Omron CX-Programmer project NewProject (CX-Programmer 9.63)

# PLC AutoAvanPLC: CJ2M CPU33
I/O table (CPU CJ2M-CPU33): rack 0 slot 0 CJ1W-ID211; rack 0 slot 1 CJ1W-OC211; rack 0 slot 11 CJ2M-EIP21

## Global symbols (name address type ; comment)
AM_ProcStatus W11 CHANNEL  ; Automatic Mode Process Status
AM_SReset W101.01 BOOL  ; Automatic Mode Shift Reset
AM_Shift W100.00 BOOL  ; Automatic Mode Shift
D22.03 BOOL  ; External Out Cilinder
W11.04 BOOL  ; .
B_Start 0.01 BOOL  ; Fisical  Start Button
C_Actual_X D14 CHANNEL  ; Actual X Postion
C_Actual_Y D15 CHANNEL  ; Actual Y Poistion
C_Clock W1.07 BOOL  ; Clock For Cartesian
C_Enable 1.06 BOOL
C_Error 0.07 BOOL  ; Fisical Cartesian Error
C_Next_X D10 CHANNEL  ; New X Position
C_Next_Y D11 CHANNEL  ; Next Y
C_Reach 0.08 BOOL  ; Fisical Cartesian Position Reached
Cartesian CartesianSimulator
DN_Pointer D97 CHANNEL  ; Pointer to the Number of Drills of Program
Drill 1.05 BOOL  ; Fisical Drill
EMERG 0.00 BOOL  ; Fisical Emergency
Ext_CEnable D22.06 BOOL  ; External Cartesian Enable
Ext_Drill D22.05 BOOL  ; External Dril
Ext_GL D22.02 BOOL  ; External Green Light
Ext_RL D22.00 BOOL  ; External Red Light
Ext_YL D22.01 BOOL  ; External Yellow Light
Ext_ZC D22.04 BOOL  ; External Z Cinder
F_AM D20.06 BOOL  ; Flag Automatic Mode
F_EM D20.07 BOOL  ; Flag End Mode
F_Incialization D20.00 BOOL  ; Flag for Incialization Process
F_MM D20.04 BOOL  ; Flag Manual Mode
F_MS D20.02 BOOL  ; Flag for Mode Selection
GL 1.02 BOOL  ; Fisical Green Light
INI_SReset W100.01 BOOL  ; Inicialization Shift Reset
INI_Shift W100.00 BOOL  ; INicialization Shift Bit
I_BStart D0.01 BOOL  ; Start Button
I_CError D0.07 BOOL  ; Cartesian Error
I_CReach D0.08 BOOL  ; Cartesian Position Reached
I_EMERG D0.00 BOOL  ; Emergency
I_SP D0.02 BOOL  ; Piece Sensor
I_a0 D0.03 BOOL  ; Z- Sensor
I_a1 D0.04 BOOL  ; Z+ Sensor
I_a2 D0.05 BOOL  ; O- Sensor
I_a3 D0.06 BOOL  ; O+ Sensor
Init_ProcStatus W10 CHANNEL  ; Inicialization Process status
Init_St0 W10.00 BOOL  ; Inicialization Stage 0
Init_St1 W10.01 BOOL  ; Inicialization Stage 1
Init_St2 W10.02 BOOL  ; Inicialization Stage 2
Init_St3 W10.03 BOOL  ; Inicialization Stage 3
M_Aux W20.01 BOOL  ; Main Process Auxiliary Flag
N_Drills D96 CHANNEL  ; Number of Drill Done
OC 1.03 BOOL  ; Fisical Out Cilinder +
O_CEnable D1.06 BOOL  ; Enable Cartesian Motor
O_Drill D1.05 BOOL  ; Drill
O_GL D1.02 BOOL  ; Green Light
O_OC D1.03 BOOL  ; Out Cilinder +
O_RL D1.00 BOOL  ; Red Light
O_YL D1.01 BOOL  ; Yellow Light
O_ZC D1.04 BOOL  ; Z Cilinder +
PN_Pointer D50 CHANNEL  ; Program Number_Pointer
RL 1.00 BOOL  ; Fisical Red Light
S_P 0.02 BOOL  ; Fisical Piece Sensor
Sct_Auto D20.05 BOOL  ; Selector Automatic Mode
Sct_Manual D20.03 BOOL  ; Select Manual Mode
Sim_C_Reach W1.00 BOOL  ; Simulation of C_Reach
StopNow W0.00 BOOL  ; StopNow
X_Pointer D98 CHANNEL  ; Pointer of Position X
YL 1.01 BOOL  ; Fisical Yellow Light
Y_Pointer D99 CHANNEL  ; Pointer of Position Y
ZC 1.04 BOOL  ; Fisical Z Cilinder +
a_0 0.03 BOOL  ; Fisical Z- Sensor
a_1 0.04 BOOL  ; Fisical Z+ Sensor
a_2 0.05 BOOL  ; Fisical O- Sensor
a_3 0.06 BOOL  ; Fisical O+ Sensor

## Program Auto_Fura (cyclic task 0)
; Auto Fura
Local symbols
DH100 CHANNEL

### Section HWInput_Output

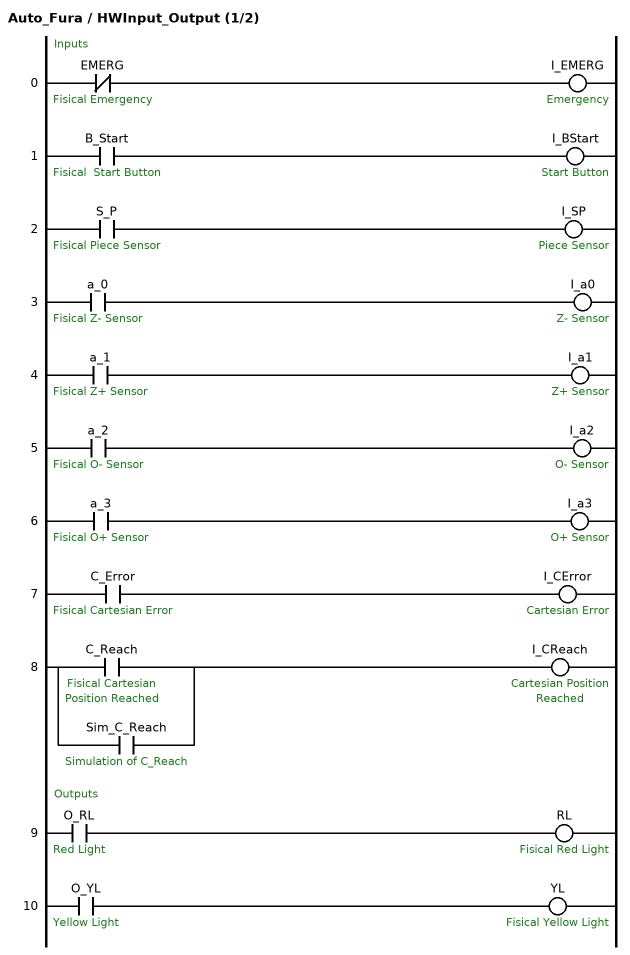
; rung 0: Inputs
LDNOT EMERG  ; Fisical Emergency
OUT I_EMERG  ; Emergency
; rung 1
LD B_Start  ; Fisical  Start Button
OUT I_BStart  ; Start Button
; rung 2
LD S_P  ; Fisical Piece Sensor
OUT I_SP  ; Piece Sensor
; rung 3
LD a_0  ; Fisical Z- Sensor
OUT I_a0  ; Z- Sensor
; rung 4
LD a_1  ; Fisical Z+ Sensor
OUT I_a1  ; Z+ Sensor
; rung 5
LD a_2  ; Fisical O- Sensor
OUT I_a2  ; O- Sensor
; rung 6
LD a_3  ; Fisical O+ Sensor
OUT I_a3  ; O+ Sensor
; rung 7
LD C_Error  ; Fisical Cartesian Error
OUT I_CError  ; Cartesian Error
; rung 8
LD C_Reach  ; Fisical Cartesian Position Reached
OR Sim_C_Reach  ; Simulation of C_Reach
OUT I_CReach  ; Cartesian Position Reached
; rung 9: Outputs
LD O_RL  ; Red Light
OUT RL  ; Fisical Red Light
; rung 10
LD O_YL  ; Yellow Light
OUT YL  ; Fisical Yellow Light

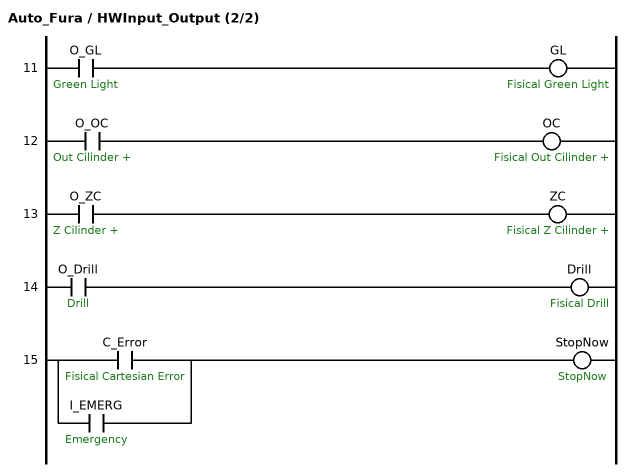
; rung 11
LD O_GL  ; Green Light
OUT GL  ; Fisical Green Light
; rung 12
LD O_OC  ; Out Cilinder +
OUT OC  ; Fisical Out Cilinder +
; rung 13
LD O_ZC  ; Z Cilinder +
OUT ZC  ; Fisical Z Cilinder +
; rung 14
LD O_Drill  ; Drill
OUT Drill  ; Fisical Drill
; rung 15
LD C_Error  ; Fisical Cartesian Error
OR I_EMERG  ; Emergency
OUT StopNow  ; StopNow

### Section Main

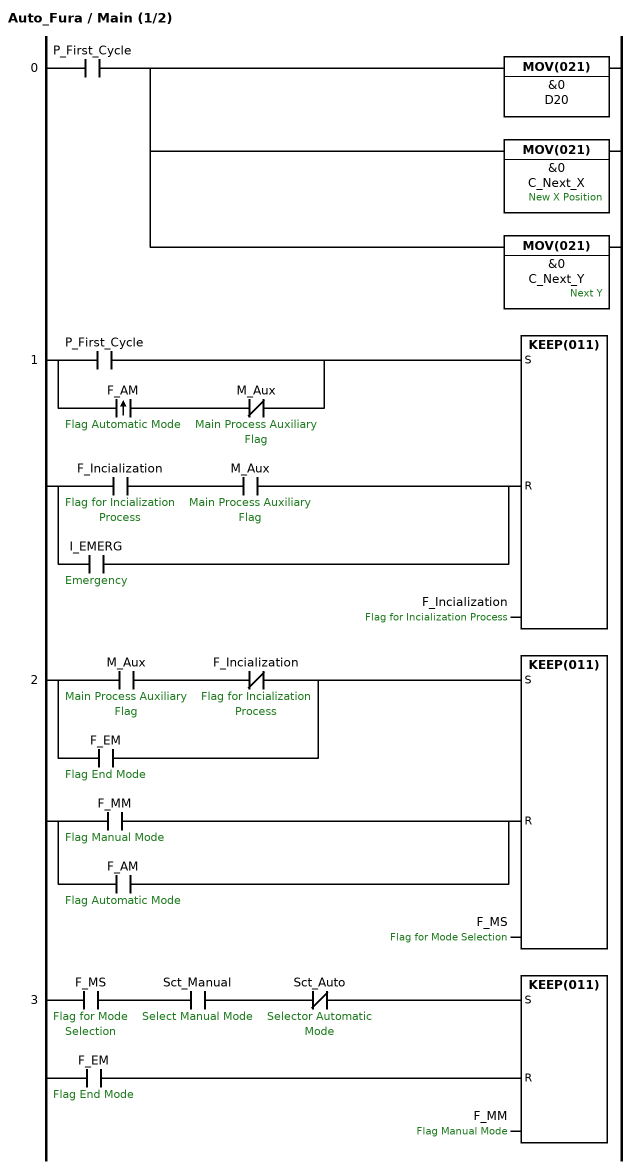
; rung 0
LD P_First_Cycle
MOV(021) &0 D20
MOV(021) &0 C_Next_X  ; New X Position
MOV(021) &0 C_Next_Y  ; Next Y
; rung 1
LD P_First_Cycle
@LD F_AM  ; Flag Automatic Mode
ANDNOT M_Aux  ; Main Process Auxiliary Flag
ORLD
LD F_Incialization  ; Flag for Incialization Process
AND M_Aux  ; Main Process Auxiliary Flag
OR I_EMERG  ; Emergency
KEEP(011) F_Incialization  ; Flag for Incialization Process
; rung 2
LD M_Aux  ; Main Process Auxiliary Flag
ANDNOT F_Incialization  ; Flag for Incialization Process
OR F_EM  ; Flag End Mode
LD F_MM  ; Flag Manual Mode
OR F_AM  ; Flag Automatic Mode
KEEP(011) F_MS  ; Flag for Mode Selection
; rung 3
LD F_MS  ; Flag for Mode Selection
AND Sct_Manual  ; Select Manual Mode
ANDNOT Sct_Auto  ; Selector Automatic Mode
LD F_EM  ; Flag End Mode
KEEP(011) F_MM  ; Flag Manual Mode

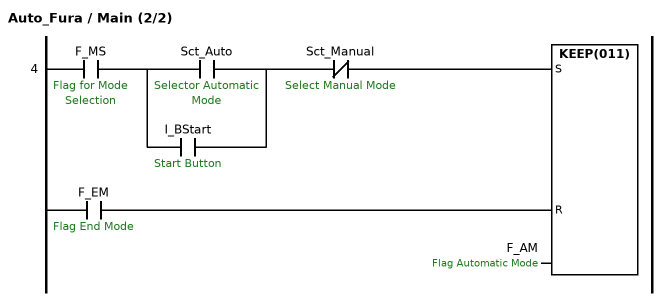
; rung 4
LD F_MS  ; Flag for Mode Selection
LD Sct_Auto  ; Selector Automatic Mode
OR I_BStart  ; Start Button
ANDLD
ANDNOT Sct_Manual  ; Select Manual Mode
LD F_EM  ; Flag End Mode
KEEP(011) F_AM  ; Flag Automatic Mode

### Section Iniciation

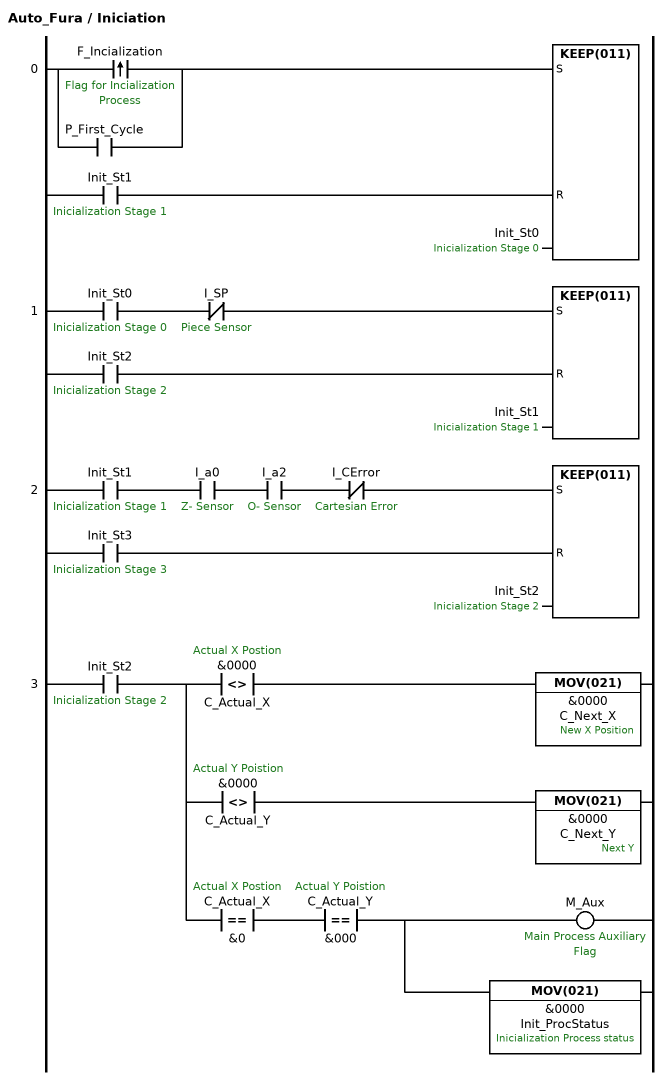
; rung 0
@LD F_Incialization  ; Flag for Incialization Process
OR P_First_Cycle
LD Init_St1  ; Inicialization Stage 1
KEEP(011) Init_St0  ; Inicialization Stage 0
; rung 1
LD Init_St0  ; Inicialization Stage 0
ANDNOT I_SP  ; Piece Sensor
LD Init_St2  ; Inicialization Stage 2
KEEP(011) Init_St1  ; Inicialization Stage 1
; rung 2
LD Init_St1  ; Inicialization Stage 1
AND I_a0  ; Z- Sensor
AND I_a2  ; O- Sensor
ANDNOT I_CError  ; Cartesian Error
LD Init_St3  ; Inicialization Stage 3
KEEP(011) Init_St2  ; Inicialization Stage 2
; rung 3
LD Init_St2  ; Inicialization Stage 2
OUT TR0
AND<>(305) &0000 C_Actual_X  ; Actual X Postion
MOV(021) &0000 C_Next_X  ; New X Position
LD TR0
AND<>(305) &0000 C_Actual_Y  ; Actual Y Poistion
MOV(021) &0000 C_Next_Y  ; Next Y
LD TR0
AND=(300) C_Actual_X &0  ; Actual X Postion
AND=(300) C_Actual_Y &000  ; Actual Y Poistion
OUT M_Aux  ; Main Process Auxiliary Flag
MOV(021) &0000 Init_ProcStatus  ; Inicialization Process status

### Section SerialCam
; Input from Camera

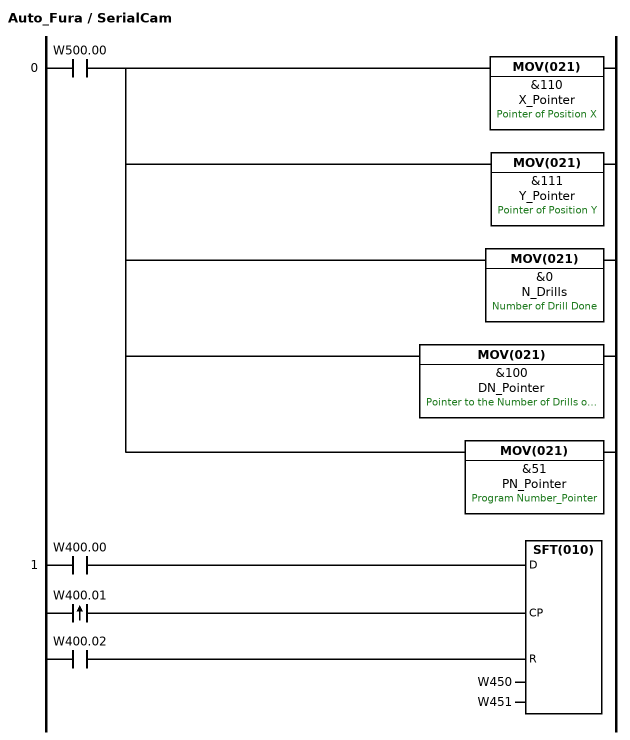
; rung 0
LD W500.00
MOV(021) &110 X_Pointer  ; Pointer of Position X
MOV(021) &111 Y_Pointer  ; Pointer of Position Y
MOV(021) &0 N_Drills  ; Number of Drill Done
MOV(021) &100 DN_Pointer  ; Pointer to the Number of Drills of Program
MOV(021) &51 PN_Pointer  ; Program Number_Pointer
; rung 1
LD W400.00
@LD W400.01
LD W400.02
SFT(010) W450 W451

### Section AutoMode

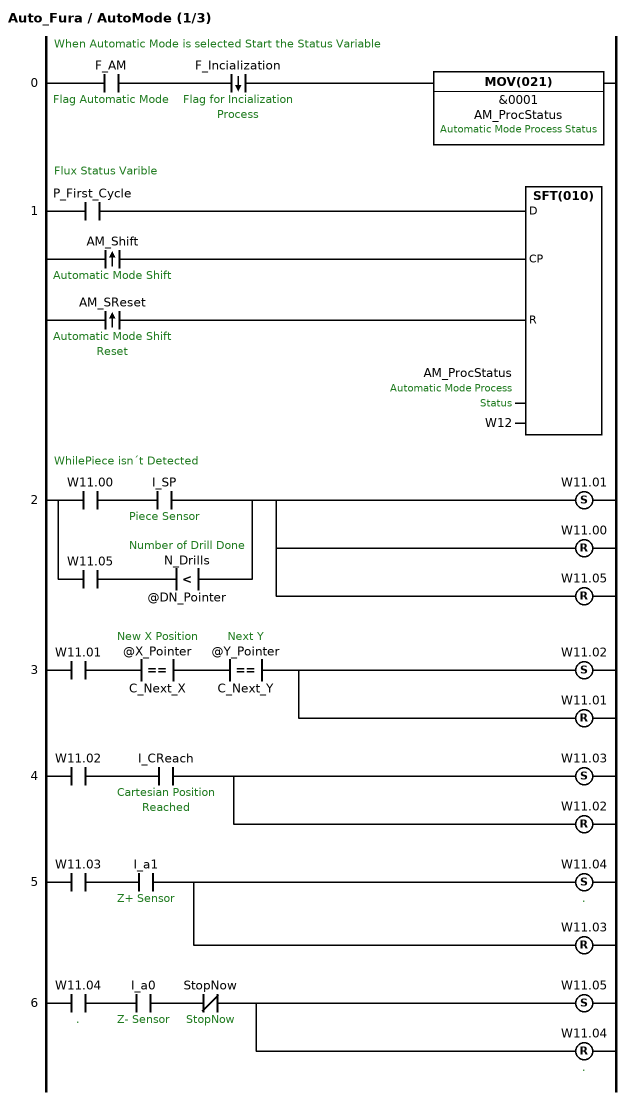
; rung 0: When Automatic Mode is selected Start the Status Variable
LD F_AM  ; Flag Automatic Mode
%AND F_Incialization  ; Flag for Incialization Process
MOV(021) &0001 AM_ProcStatus  ; Automatic Mode Process Status
; rung 1: Flux Status Varible
LD P_First_Cycle
@LD AM_Shift  ; Automatic Mode Shift
@LD AM_SReset  ; Automatic Mode Shift Reset
SFT(010) AM_ProcStatus W12  ; Automatic Mode Process Status
; rung 2: WhilePiece isn´t Detected
LD W11.00
AND I_SP  ; Piece Sensor
LD W11.05
AND<(310) N_Drills @DN_Pointer  ; Number of Drill Done
ORLD
SET W11.01
RSET W11.00
RSET W11.05
; rung 3
LD W11.01
AND=(300) @X_Pointer C_Next_X  ; New X Position
AND=(300) @Y_Pointer C_Next_Y  ; Next Y
SET W11.02
RSET W11.01
; rung 4
LD W11.02
AND I_CReach  ; Cartesian Position Reached
SET W11.03
RSET W11.02
; rung 5
LD W11.03
AND I_a1  ; Z+ Sensor
SET W11.04  ; .
RSET W11.03
; rung 6
LD W11.04  ; .
AND I_a0  ; Z- Sensor
ANDNOT StopNow  ; StopNow
SET W11.05
RSET W11.04  ; .

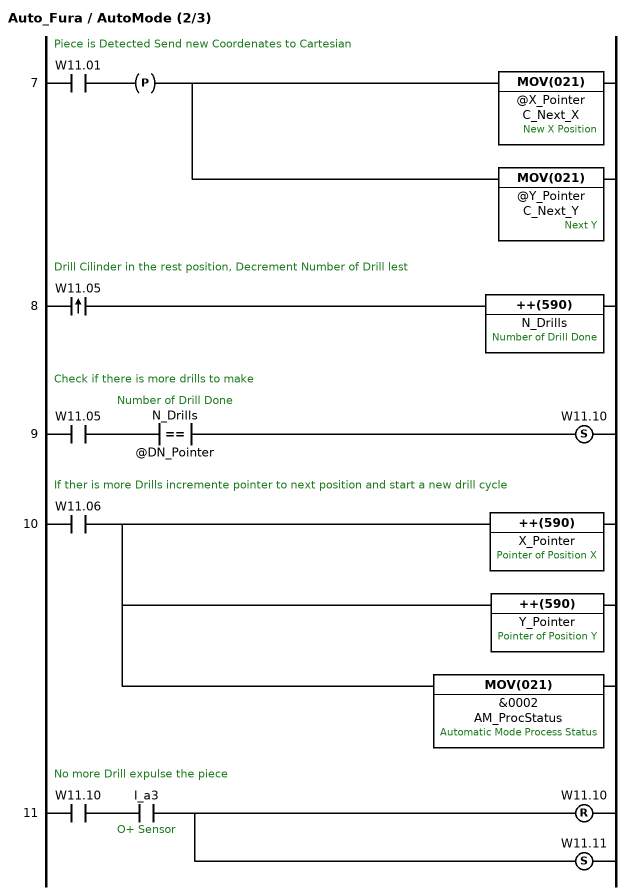
; rung 7: Piece is Detected Send new Coordenates to Cartesian
LD W11.01
UP(521)
MOV(021) @X_Pointer C_Next_X  ; New X Position
MOV(021) @Y_Pointer C_Next_Y  ; Next Y
; rung 8: Drill Cilinder in the rest position, Decrement Number of Drill lest
@LD W11.05
++(590) N_Drills  ; Number of Drill Done
; rung 9: Check if there is more drills to make
LD W11.05
AND=(300) N_Drills @DN_Pointer  ; Number of Drill Done
SET W11.10
; rung 10: If ther is more Drills incremente pointer to next position and start a new drill cycle
LD W11.06
++(590) X_Pointer  ; Pointer of Position X
++(590) Y_Pointer  ; Pointer of Position Y
MOV(021) &0002 AM_ProcStatus  ; Automatic Mode Process Status
; rung 11: No more Drill expulse the piece
LD W11.10
AND I_a3  ; O+ Sensor
RSET W11.10
SET W11.11

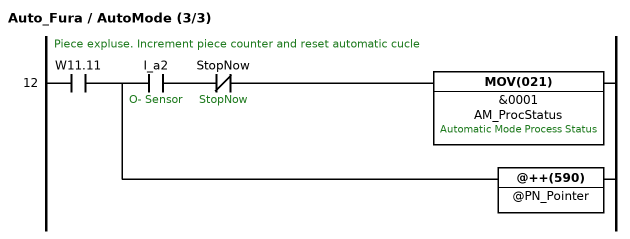
; rung 12: Piece expluse. Increment piece counter and reset automatic cucle
LD W11.11
OUT TR0
AND I_a2  ; O- Sensor
ANDNOT StopNow  ; StopNow
MOV(021) &0001 AM_ProcStatus  ; Automatic Mode Process Status
LD TR0
@++(590) @PN_Pointer

### Section ManualMode

### Section Output

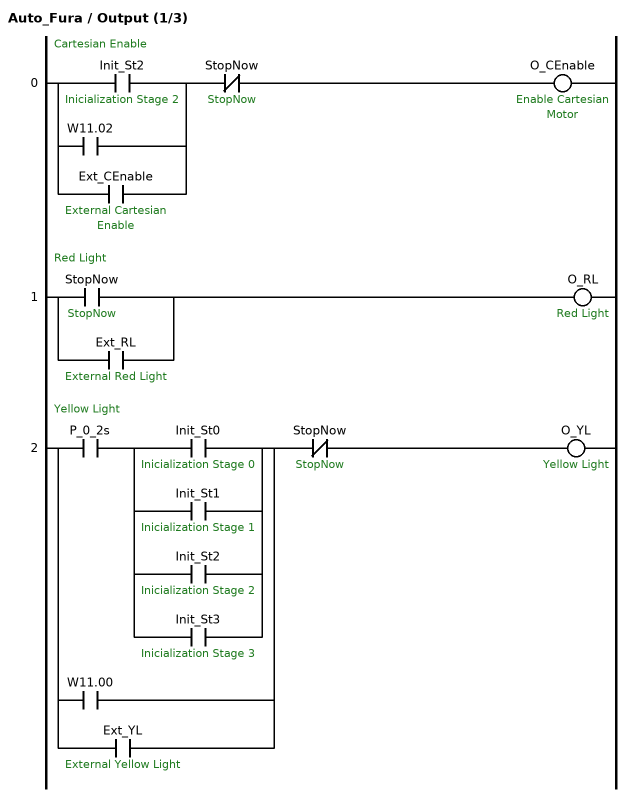
; rung 0: Cartesian Enable
LD Init_St2  ; Inicialization Stage 2
OR W11.02
OR Ext_CEnable  ; External Cartesian Enable
ANDNOT StopNow  ; StopNow
OUT O_CEnable  ; Enable Cartesian Motor
; rung 1: Red Light
LD StopNow  ; StopNow
OR Ext_RL  ; External Red Light
OUT O_RL  ; Red Light
; rung 2: Yellow Light
LD P_0_2s
LD Init_St0  ; Inicialization Stage 0
OR Init_St1  ; Inicialization Stage 1
OR Init_St2  ; Inicialization Stage 2
OR Init_St3  ; Inicialization Stage 3
ANDLD
OR W11.00
OR Ext_YL  ; External Yellow Light
ANDNOT StopNow  ; StopNow
OUT O_YL  ; Yellow Light

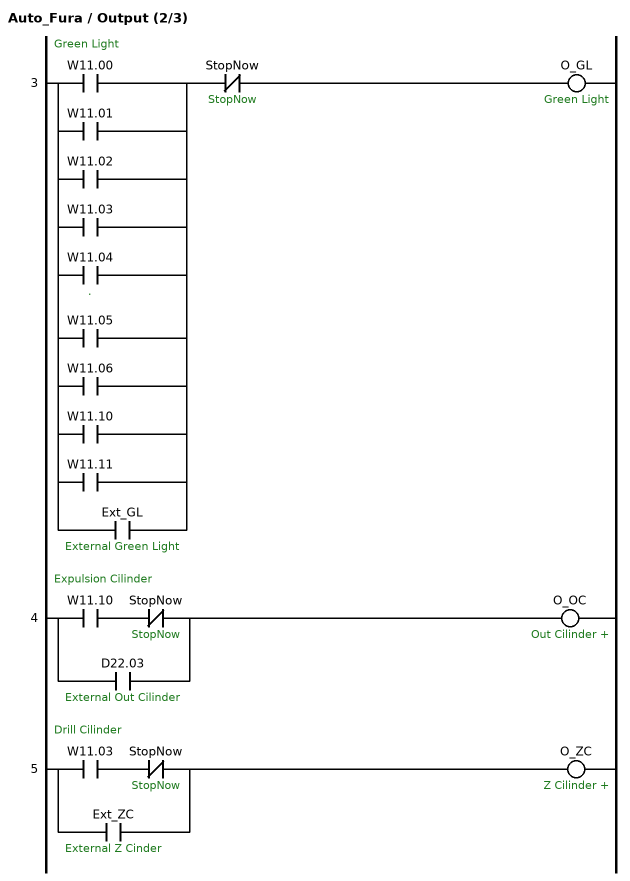
; rung 3: Green Light
LD W11.00
OR W11.01
OR W11.02
OR W11.03
OR W11.04  ; .
OR W11.05
OR W11.06
OR W11.10
OR W11.11
OR Ext_GL  ; External Green Light
ANDNOT StopNow  ; StopNow
OUT O_GL  ; Green Light
; rung 4: Expulsion Cilinder
LD W11.10
ANDNOT StopNow  ; StopNow
OR D22.03  ; External Out Cilinder
OUT O_OC  ; Out Cilinder +
; rung 5: Drill Cilinder
LD W11.03
ANDNOT StopNow  ; StopNow
OR Ext_ZC  ; External Z Cinder
OUT O_ZC  ; Z Cilinder +

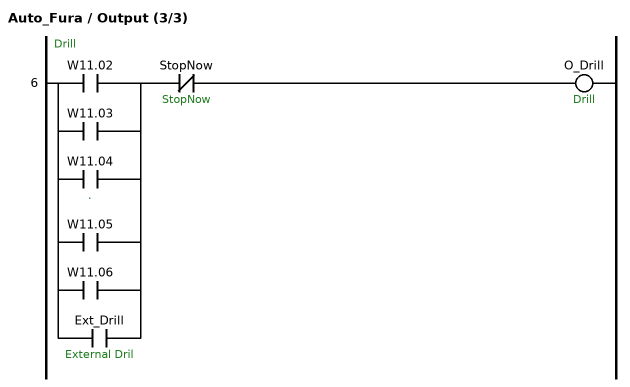
; rung 6: Drill
LD W11.02
OR W11.03
OR W11.04  ; .
OR W11.05
OR W11.06
OR Ext_Drill  ; External Dril
ANDNOT StopNow  ; StopNow
OUT O_Drill  ; Drill

### Section CartesianControl
; Cartesian Simulator

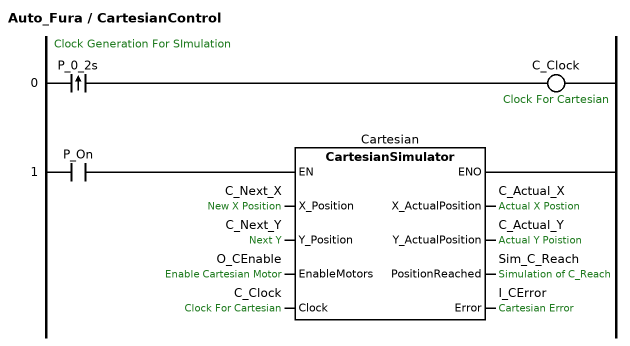
; rung 0: Clock Generation For SImulation
@LD P_0_2s
OUT C_Clock  ; Clock For Cartesian
; rung 1
LD P_On
CALL Cartesian : CartesianSimulator (X_Position := C_Next_X, Y_Position := C_Next_Y, EnableMotors := O_CEnable, Clock := C_Clock, X_ActualPosition => C_Actual_X, Y_ActualPosition => C_Actual_Y, PositionReached => Sim_C_Reach, Error => I_CError)  ; New X Position, Next Y, Enable Cartesian Motor, Clock For Cartesian, Actual X Postion, Actual Y Poistion, Simulation of C_Reach, Cartesian Error

### Section EthernetInterface

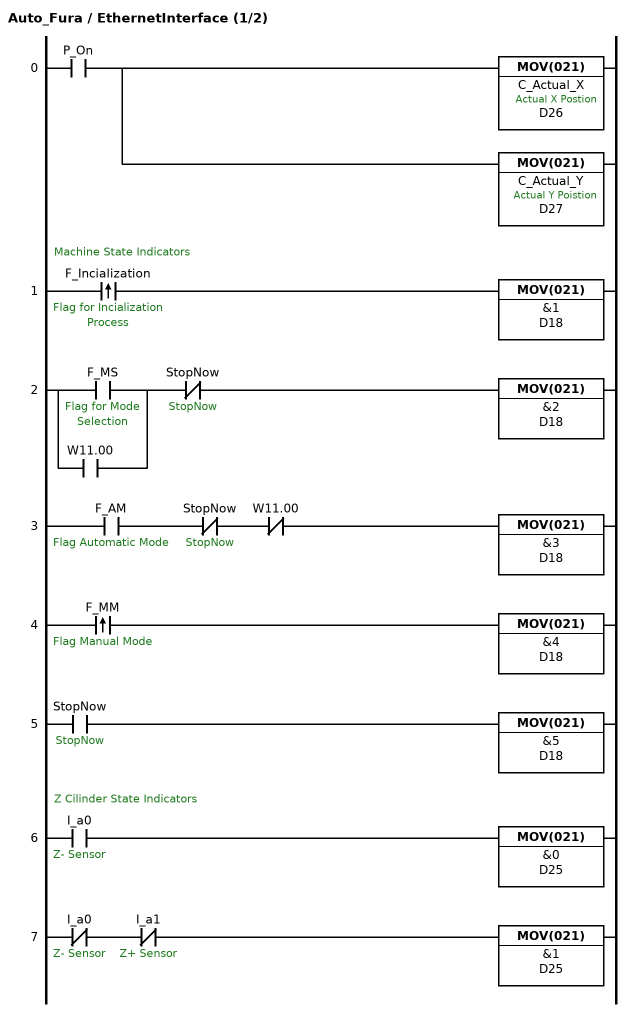
; rung 0
LD P_On
MOV(021) C_Actual_X D26  ; Actual X Postion
MOV(021) C_Actual_Y D27  ; Actual Y Poistion
; rung 1: Machine State Indicators
@LD F_Incialization  ; Flag for Incialization Process
MOV(021) &1 D18
; rung 2
LD F_MS  ; Flag for Mode Selection
OR W11.00
ANDNOT StopNow  ; StopNow
MOV(021) &2 D18
; rung 3
LD F_AM  ; Flag Automatic Mode
ANDNOT StopNow  ; StopNow
ANDNOT W11.00
MOV(021) &3 D18
; rung 4
@LD F_MM  ; Flag Manual Mode
MOV(021) &4 D18
; rung 5
LD StopNow  ; StopNow
MOV(021) &5 D18
; rung 6: Z Cilinder State Indicators
LD I_a0  ; Z- Sensor
MOV(021) &0 D25
; rung 7
LDNOT I_a0  ; Z- Sensor
ANDNOT I_a1  ; Z+ Sensor
MOV(021) &1 D25

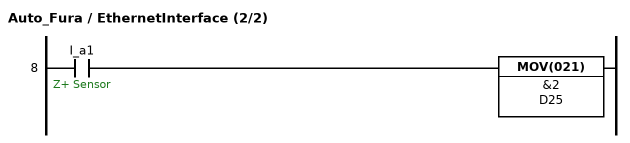
; rung 8
LD I_a1  ; Z+ Sensor
MOV(021) &2 D25

### Section END
; rung 0
END(001)

## Function block CartesianSimulator
VAR_INPUT
  X_Position : INT;
  Y_Position : INT;
  EnableMotors : BOOL;
  Clock : BOOL;
END_VAR
VAR_OUTPUT
  X_ActualPosition : INT;
  Y_ActualPosition : INT;
  PositionReached : BOOL;
  Error : BOOL;
END_VAR
VAR
  XCounter : INT;
  YCounter : INT;
  errorCounter : INT;
END_VAR
XCounter := X_ActualPosition;
YCounter := Y_ActualPosition;

IF (X_Position > 1500) OR (Y_Position > 1500) THEN
	Error := TRUE;
	
ELSE
	
	IF Error = FALSE THEN
			IF (XCounter <> X_Position) or (YCounter <> Y_Position) THEN
			
			IF XCounter < X_Position THEN
				IF (Clock = TRUE) AND (EnableMotors = TRUE) THEN
					XCounter := XCounter + 1;
					errorCounter:= errorCounter+1;
				END_IF;
			END_IF;

			IF XCounter > X_Position THEN
				IF (Clock = TRUE) AND (EnableMotors = TRUE) THEN
					XCounter := XCounter - 1;
					errorCounter:= errorCounter+1;
				END_IF;
			END_IF;
			
			X_ActualPosition := XCounter;


			IF YCounter < Y_Position THEN
				IF (Clock = TRUE) AND (EnableMotors = TRUE) THEN
					YCounter := YCounter + 1;
					errorCounter:= errorCounter+1;
				END_IF;
			END_IF;

			IF Y_ActualPosition > Y_Position THEN
				IF (Clock = TRUE) AND (EnableMotors = TRUE) THEN
					YCounter := YCounter - 1;
					errorCounter:= errorCounter+1;
				END_IF;
			END_IF;
			
			Y_ActualPosition := YCounter;

		END_IF;;

		IF (X_ActualPosition = X_Position) AND (Y_ActualPosition = Y_Position) THEN
			PositionReached := TRUE;
			errorCounter:= 0;
			
		ELSE
			PositionReached := FALSE;
			
			IF errorCounter > 1501 THEN
				Error:= TRUE;
			ELSE
				
				Error:= FALSE;
			END_IF;
			
		END_IF;
	END_IF;
	
END_IF;

IF EnableMotors = FALSE THEN
	Error:= FALSE;
	
END_IF;